ABB RAPID module: 0026CD4A

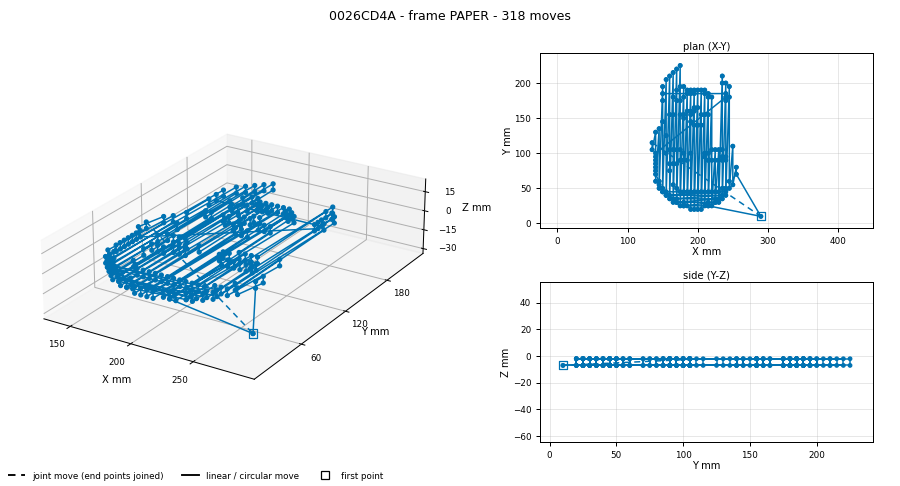
[picture p0: tool path of 0026CD4A in frame PAPER, 318 of 318 moves have a stored position in this frame; points joined in program order, loops and branches not executed]
MODULE Module1
    CONST robtarget Target_drawing_origin:=[[290,10,-2],[1,0,0,0],[0,0,0,0],[9E+09,9E+09,9E+09,9E+09,9E+09,9E+09]];


! Main procedure
PROC main()


! Clean
SetDO Do_Clean, 1;
SetDO Do_Clean, 0;
SetDO Do_Kreslit_OFF, 1;
SetDO Do_Kreslit_ON, 0;
! Draw grey
MoveJ Offs(Target_drawing_origin,0,0,-5),v100,fine,PencilHolder\WObj:=PAPER;
MoveL Offs(Target_drawing_origin,-35,60,-5),v100,fine,PencilHolder\WObj:=PAPER;
WaitRob \InPos;
MoveL Offs(Target_drawing_origin,-35,60,0),v100,fine,PencilHolder\WObj:=PAPER;
WaitRob \InPos;
SetDO Do_Kreslit_ON, 1;
SetDO Do_Kreslit_OFF, 0;
MoveL Offs(Target_drawing_origin,-35,70,0),v100,fine,PencilHolder\WObj:=PAPER;
WaitRob \InPos;
SetDO Do_Kreslit_ON, 0;
SetDO Do_Kreslit_OFF, 1;
MoveL Offs(Target_drawing_origin,-35,70,-5),v100,fine,PencilHolder\WObj:=PAPER;
WaitRob \InPos;
MoveL Offs(Target_drawing_origin,-40,45,-5),v100,fine,PencilHolder\WObj:=PAPER;
WaitRob \InPos;
MoveL Offs(Target_drawing_origin,-40,45,0),v100,fine,PencilHolder\WObj:=PAPER;
WaitRob \InPos;
SetDO Do_Kreslit_ON, 1;
SetDO Do_Kreslit_OFF, 0;
MoveL Offs(Target_drawing_origin,-40,100,0),v100,fine,PencilHolder\WObj:=PAPER;
WaitRob \InPos;
SetDO Do_Kreslit_ON, 0;
SetDO Do_Kreslit_OFF, 1;
MoveL Offs(Target_drawing_origin,-40,100,-5),v100,fine,PencilHolder\WObj:=PAPER;
WaitRob \InPos;
MoveL Offs(Target_drawing_origin,-45,40,-5),v100,fine,PencilHolder\WObj:=PAPER;
WaitRob \InPos;
MoveL Offs(Target_drawing_origin,-45,40,0),v100,fine,PencilHolder\WObj:=PAPER;
WaitRob \InPos;
SetDO Do_Kreslit_ON, 1;
SetDO Do_Kreslit_OFF, 0;
MoveL Offs(Target_drawing_origin,-45,50,0),v100,fine,PencilHolder\WObj:=PAPER;
WaitRob \InPos;
SetDO Do_Kreslit_ON, 0;
SetDO Do_Kreslit_OFF, 1;
MoveL Offs(Target_drawing_origin,-45,50,-5),v100,fine,PencilHolder\WObj:=PAPER;
WaitRob \InPos;
MoveL Offs(Target_drawing_origin,-45,170,-5),v100,fine,PencilHolder\WObj:=PAPER;
WaitRob \InPos;
MoveL Offs(Target_drawing_origin,-45,170,0),v100,fine,PencilHolder\WObj:=PAPER;
WaitRob \InPos;
SetDO Do_Kreslit_ON, 1;
SetDO Do_Kreslit_OFF, 0;
MoveL Offs(Target_drawing_origin,-45,185,0),v100,fine,PencilHolder\WObj:=PAPER;
WaitRob \InPos;
SetDO Do_Kreslit_ON, 0;
SetDO Do_Kreslit_OFF, 1;
MoveL Offs(Target_drawing_origin,-45,185,-5),v100,fine,PencilHolder\WObj:=PAPER;
WaitRob \InPos;
MoveL Offs(Target_drawing_origin,-50,30,-5),v100,fine,PencilHolder\WObj:=PAPER;
WaitRob \InPos;
MoveL Offs(Target_drawing_origin,-50,30,0),v100,fine,PencilHolder\WObj:=PAPER;
WaitRob \InPos;
SetDO Do_Kreslit_ON, 1;
SetDO Do_Kreslit_OFF, 0;
MoveL Offs(Target_drawing_origin,-50,40,0),v100,fine,PencilHolder\WObj:=PAPER;
WaitRob \InPos;
SetDO Do_Kreslit_ON, 0;
SetDO Do_Kreslit_OFF, 1;
MoveL Offs(Target_drawing_origin,-50,40,-5),v100,fine,PencilHolder\WObj:=PAPER;
WaitRob \InPos;
MoveL Offs(Target_drawing_origin,-50,80,-5),v100,fine,PencilHolder\WObj:=PAPER;
WaitRob \InPos;
MoveL Offs(Target_drawing_origin,-50,80,0),v100,fine,PencilHolder\WObj:=PAPER;
WaitRob \InPos;
SetDO Do_Kreslit_ON, 1;
SetDO Do_Kreslit_OFF, 0;
MoveL Offs(Target_drawing_origin,-50,85,0),v100,fine,PencilHolder\WObj:=PAPER;
WaitRob \InPos;
SetDO Do_Kreslit_ON, 0;
SetDO Do_Kreslit_OFF, 1;
MoveL Offs(Target_drawing_origin,-50,85,-5),v100,fine,PencilHolder\WObj:=PAPER;
WaitRob \InPos;
MoveL Offs(Target_drawing_origin,-50,165,-5),v100,fine,PencilHolder\WObj:=PAPER;
WaitRob \InPos;
MoveL Offs(Target_drawing_origin,-50,165,0),v100,fine,PencilHolder\WObj:=PAPER;
WaitRob \InPos;
SetDO Do_Kreslit_ON, 1;
SetDO Do_Kreslit_OFF, 0;
MoveL Offs(Target_drawing_origin,-50,190,0),v100,fine,PencilHolder\WObj:=PAPER;
WaitRob \InPos;
SetDO Do_Kreslit_ON, 0;
SetDO Do_Kreslit_OFF, 1;
MoveL Offs(Target_drawing_origin,-50,190,-5),v100,fine,PencilHolder\WObj:=PAPER;
WaitRob \InPos;
MoveL Offs(Target_drawing_origin,-55,25,-5),v100,fine,PencilHolder\WObj:=PAPER;
WaitRob \InPos;
MoveL Offs(Target_drawing_origin,-55,25,0),v100,fine,PencilHolder\WObj:=PAPER;
WaitRob \InPos;
SetDO Do_Kreslit_ON, 1;
SetDO Do_Kreslit_OFF, 0;
MoveL Offs(Target_drawing_origin,-55,40,0),v100,fine,PencilHolder\WObj:=PAPER;
WaitRob \InPos;
SetDO Do_Kreslit_ON, 0;
SetDO Do_Kreslit_OFF, 1;
MoveL Offs(Target_drawing_origin,-55,40,-5),v100,fine,PencilHolder\WObj:=PAPER;
WaitRob \InPos;
MoveL Offs(Target_drawing_origin,-55,80,-5),v100,fine,PencilHolder\WObj:=PAPER;
WaitRob \InPos;
MoveL Offs(Target_drawing_origin,-55,80,0),v100,fine,PencilHolder\WObj:=PAPER;
WaitRob \InPos;
SetDO Do_Kreslit_ON, 1;
SetDO Do_Kreslit_OFF, 0;
MoveL Offs(Target_drawing_origin,-55,85,0),v100,fine,PencilHolder\WObj:=PAPER;
WaitRob \InPos;
SetDO Do_Kreslit_ON, 0;
SetDO Do_Kreslit_OFF, 1;
MoveL Offs(Target_drawing_origin,-55,85,-5),v100,fine,PencilHolder\WObj:=PAPER;
WaitRob \InPos;
MoveL Offs(Target_drawing_origin,-55,95,-5),v100,fine,PencilHolder\WObj:=PAPER;
WaitRob \InPos;
MoveL Offs(Target_drawing_origin,-55,95,0),v100,fine,PencilHolder\WObj:=PAPER;
WaitRob \InPos;
SetDO Do_Kreslit_ON, 1;
SetDO Do_Kreslit_OFF, 0;
MoveL Offs(Target_drawing_origin,-55,190,0),v100,fine,PencilHolder\WObj:=PAPER;
WaitRob \InPos;
SetDO Do_Kreslit_ON, 0;
SetDO Do_Kreslit_OFF, 1;
MoveL Offs(Target_drawing_origin,-55,190,-5),v100,fine,PencilHolder\WObj:=PAPER;
WaitRob \InPos;
MoveL Offs(Target_drawing_origin,-55,200,-5),v100,fine,PencilHolder\WObj:=PAPER;
WaitRob \InPos;
MoveL Offs(Target_drawing_origin,-55,200,0),v100,fine,PencilHolder\WObj:=PAPER;
WaitRob \InPos;
SetDO Do_Kreslit_ON, 1;
SetDO Do_Kreslit_OFF, 0;
MoveL Offs(Target_drawing_origin,-60,20,0),v100,fine,PencilHolder\WObj:=PAPER;
WaitRob \InPos;
SetDO Do_Kreslit_ON, 0;
SetDO Do_Kreslit_OFF, 1;
MoveL Offs(Target_drawing_origin,-60,20,-5),v100,fine,PencilHolder\WObj:=PAPER;
WaitRob \InPos;
MoveL Offs(Target_drawing_origin,-60,35,-5),v100,fine,PencilHolder\WObj:=PAPER;
WaitRob \InPos;
MoveL Offs(Target_drawing_origin,-60,35,0),v100,fine,PencilHolder\WObj:=PAPER;
WaitRob \InPos;
SetDO Do_Kreslit_ON, 1;
SetDO Do_Kreslit_OFF, 0;
MoveL Offs(Target_drawing_origin,-60,80,0),v100,fine,PencilHolder\WObj:=PAPER;
WaitRob \InPos;
SetDO Do_Kreslit_ON, 0;
SetDO Do_Kreslit_OFF, 1;
MoveL Offs(Target_drawing_origin,-60,80,-5),v100,fine,PencilHolder\WObj:=PAPER;
WaitRob \InPos;
MoveL Offs(Target_drawing_origin,-60,95,-5),v100,fine,PencilHolder\WObj:=PAPER;
WaitRob \InPos;
MoveL Offs(Target_drawing_origin,-60,95,0),v100,fine,PencilHolder\WObj:=PAPER;
WaitRob \InPos;
SetDO Do_Kreslit_ON, 1;
SetDO Do_Kreslit_OFF, 0;
MoveL Offs(Target_drawing_origin,-65,20,0),v100,fine,PencilHolder\WObj:=PAPER;
WaitRob \InPos;
SetDO Do_Kreslit_ON, 0;
SetDO Do_Kreslit_OFF, 1;
MoveL Offs(Target_drawing_origin,-65,20,-5),v100,fine,PencilHolder\WObj:=PAPER;
WaitRob \InPos;
MoveL Offs(Target_drawing_origin,-65,35,-5),v100,fine,PencilHolder\WObj:=PAPER;
WaitRob \InPos;
MoveL Offs(Target_drawing_origin,-65,35,0),v100,fine,PencilHolder\WObj:=PAPER;
WaitRob \InPos;
SetDO Do_Kreslit_ON, 1;
SetDO Do_Kreslit_OFF, 0;
MoveL Offs(Target_drawing_origin,-65,80,0),v100,fine,PencilHolder\WObj:=PAPER;
WaitRob \InPos;
SetDO Do_Kreslit_ON, 0;
SetDO Do_Kreslit_OFF, 1;
MoveL Offs(Target_drawing_origin,-65,80,-5),v100,fine,PencilHolder\WObj:=PAPER;
WaitRob \InPos;
MoveL Offs(Target_drawing_origin,-65,95,-5),v100,fine,PencilHolder\WObj:=PAPER;
WaitRob \InPos;
MoveL Offs(Target_drawing_origin,-65,95,0),v100,fine,PencilHolder\WObj:=PAPER;
WaitRob \InPos;
SetDO Do_Kreslit_ON, 1;
SetDO Do_Kreslit_OFF, 0;
MoveL Offs(Target_drawing_origin,-70,15,0),v100,fine,PencilHolder\WObj:=PAPER;
WaitRob \InPos;
SetDO Do_Kreslit_ON, 0;
SetDO Do_Kreslit_OFF, 1;
MoveL Offs(Target_drawing_origin,-70,15,-5),v100,fine,PencilHolder\WObj:=PAPER;
WaitRob \InPos;
MoveL Offs(Target_drawing_origin,-70,35,-5),v100,fine,PencilHolder\WObj:=PAPER;
WaitRob \InPos;
MoveL Offs(Target_drawing_origin,-70,35,0),v100,fine,PencilHolder\WObj:=PAPER;
WaitRob \InPos;
SetDO Do_Kreslit_ON, 1;
SetDO Do_Kreslit_OFF, 0;
MoveL Offs(Target_drawing_origin,-70,80,0),v100,fine,PencilHolder\WObj:=PAPER;
WaitRob \InPos;
SetDO Do_Kreslit_ON, 0;
SetDO Do_Kreslit_OFF, 1;
MoveL Offs(Target_drawing_origin,-70,80,-5),v100,fine,PencilHolder\WObj:=PAPER;
WaitRob \InPos;
MoveL Offs(Target_drawing_origin,-70,95,-5),v100,fine,PencilHolder\WObj:=PAPER;
WaitRob \InPos;
MoveL Offs(Target_drawing_origin,-70,95,0),v100,fine,PencilHolder\WObj:=PAPER;
WaitRob \InPos;
SetDO Do_Kreslit_ON, 1;
SetDO Do_Kreslit_OFF, 0;
MoveL Offs(Target_drawing_origin,-70,170,0),v100,fine,PencilHolder\WObj:=PAPER;
WaitRob \InPos;
SetDO Do_Kreslit_ON, 0;
SetDO Do_Kreslit_OFF, 1;
MoveL Offs(Target_drawing_origin,-70,170,-5),v100,fine,PencilHolder\WObj:=PAPER;
WaitRob \InPos;
MoveL Offs(Target_drawing_origin,-75,15,-5),v100,fine,PencilHolder\WObj:=PAPER;
WaitRob \InPos;
MoveL Offs(Target_drawing_origin,-75,15,0),v100,fine,PencilHolder\WObj:=PAPER;
WaitRob \InPos;
SetDO Do_Kreslit_ON, 1;
SetDO Do_Kreslit_OFF, 0;
MoveL Offs(Target_drawing_origin,-75,35,0),v100,fine,PencilHolder\WObj:=PAPER;
WaitRob \InPos;
SetDO Do_Kreslit_ON, 0;
SetDO Do_Kreslit_OFF, 1;
MoveL Offs(Target_drawing_origin,-75,35,-5),v100,fine,PencilHolder\WObj:=PAPER;
WaitRob \InPos;
MoveL Offs(Target_drawing_origin,-75,80,-5),v100,fine,PencilHolder\WObj:=PAPER;
WaitRob \InPos;
MoveL Offs(Target_drawing_origin,-75,80,0),v100,fine,PencilHolder\WObj:=PAPER;
WaitRob \InPos;
SetDO Do_Kreslit_ON, 1;
SetDO Do_Kreslit_OFF, 0;
MoveL Offs(Target_drawing_origin,-75,90,0),v100,fine,PencilHolder\WObj:=PAPER;
WaitRob \InPos;
SetDO Do_Kreslit_ON, 0;
SetDO Do_Kreslit_OFF, 1;
MoveL Offs(Target_drawing_origin,-75,90,-5),v100,fine,PencilHolder\WObj:=PAPER;
WaitRob \InPos;
MoveL Offs(Target_drawing_origin,-75,145,-5),v100,fine,PencilHolder\WObj:=PAPER;
WaitRob \InPos;
MoveL Offs(Target_drawing_origin,-75,145,0),v100,fine,PencilHolder\WObj:=PAPER;
WaitRob \InPos;
SetDO Do_Kreslit_ON, 1;
SetDO Do_Kreslit_OFF, 0;
MoveL Offs(Target_drawing_origin,-75,170,0),v100,fine,PencilHolder\WObj:=PAPER;
WaitRob \InPos;
SetDO Do_Kreslit_ON, 0;
SetDO Do_Kreslit_OFF, 1;
MoveL Offs(Target_drawing_origin,-75,170,-5),v100,fine,PencilHolder\WObj:=PAPER;
WaitRob \InPos;
MoveL Offs(Target_drawing_origin,-75,175,-5),v100,fine,PencilHolder\WObj:=PAPER;
WaitRob \InPos;
MoveL Offs(Target_drawing_origin,-75,175,0),v100,fine,PencilHolder\WObj:=PAPER;
WaitRob \InPos;
SetDO Do_Kreslit_ON, 1;
SetDO Do_Kreslit_OFF, 0;
MoveL Offs(Target_drawing_origin,-80,15,0),v100,fine,PencilHolder\WObj:=PAPER;
WaitRob \InPos;
SetDO Do_Kreslit_ON, 0;
SetDO Do_Kreslit_OFF, 1;
MoveL Offs(Target_drawing_origin,-80,15,-5),v100,fine,PencilHolder\WObj:=PAPER;
WaitRob \InPos;
MoveL Offs(Target_drawing_origin,-80,35,-5),v100,fine,PencilHolder\WObj:=PAPER;
WaitRob \InPos;
MoveL Offs(Target_drawing_origin,-80,35,0),v100,fine,PencilHolder\WObj:=PAPER;
WaitRob \InPos;
SetDO Do_Kreslit_ON, 1;
SetDO Do_Kreslit_OFF, 0;
MoveL Offs(Target_drawing_origin,-80,85,0),v100,fine,PencilHolder\WObj:=PAPER;
WaitRob \InPos;
SetDO Do_Kreslit_ON, 0;
SetDO Do_Kreslit_OFF, 1;
MoveL Offs(Target_drawing_origin,-80,85,-5),v100,fine,PencilHolder\WObj:=PAPER;
WaitRob \InPos;
MoveL Offs(Target_drawing_origin,-80,90,-5),v100,fine,PencilHolder\WObj:=PAPER;
WaitRob \InPos;
MoveL Offs(Target_drawing_origin,-80,90,0),v100,fine,PencilHolder\WObj:=PAPER;
WaitRob \InPos;
SetDO Do_Kreslit_ON, 1;
SetDO Do_Kreslit_OFF, 0;
MoveL Offs(Target_drawing_origin,-80,145,0),v100,fine,PencilHolder\WObj:=PAPER;
WaitRob \InPos;
SetDO Do_Kreslit_ON, 0;
SetDO Do_Kreslit_OFF, 1;
MoveL Offs(Target_drawing_origin,-80,145,-5),v100,fine,PencilHolder\WObj:=PAPER;
WaitRob \InPos;
MoveL Offs(Target_drawing_origin,-80,175,-5),v100,fine,PencilHolder\WObj:=PAPER;
WaitRob \InPos;
MoveL Offs(Target_drawing_origin,-80,175,0),v100,fine,PencilHolder\WObj:=PAPER;
WaitRob \InPos;
SetDO Do_Kreslit_ON, 1;
SetDO Do_Kreslit_OFF, 0;
MoveL Offs(Target_drawing_origin,-80,180,0),v100,fine,PencilHolder\WObj:=PAPER;
WaitRob \InPos;
SetDO Do_Kreslit_ON, 0;
SetDO Do_Kreslit_OFF, 1;
MoveL Offs(Target_drawing_origin,-80,180,-5),v100,fine,PencilHolder\WObj:=PAPER;
WaitRob \InPos;
MoveL Offs(Target_drawing_origin,-85,10,-5),v100,fine,PencilHolder\WObj:=PAPER;
WaitRob \InPos;
MoveL Offs(Target_drawing_origin,-85,10,0),v100,fine,PencilHolder\WObj:=PAPER;
WaitRob \InPos;
SetDO Do_Kreslit_ON, 1;
SetDO Do_Kreslit_OFF, 0;
MoveL Offs(Target_drawing_origin,-85,35,0),v100,fine,PencilHolder\WObj:=PAPER;
WaitRob \InPos;
SetDO Do_Kreslit_ON, 0;
SetDO Do_Kreslit_OFF, 1;
MoveL Offs(Target_drawing_origin,-85,35,-5),v100,fine,PencilHolder\WObj:=PAPER;
WaitRob \InPos;
MoveL Offs(Target_drawing_origin,-85,130,-5),v100,fine,PencilHolder\WObj:=PAPER;
WaitRob \InPos;
MoveL Offs(Target_drawing_origin,-85,130,0),v100,fine,PencilHolder\WObj:=PAPER;
WaitRob \InPos;
SetDO Do_Kreslit_ON, 1;
SetDO Do_Kreslit_OFF, 0;
MoveL Offs(Target_drawing_origin,-85,145,0),v100,fine,PencilHolder\WObj:=PAPER;
WaitRob \InPos;
SetDO Do_Kreslit_ON, 0;
SetDO Do_Kreslit_OFF, 1;
MoveL Offs(Target_drawing_origin,-85,145,-5),v100,fine,PencilHolder\WObj:=PAPER;
WaitRob \InPos;
MoveL Offs(Target_drawing_origin,-85,180,-5),v100,fine,PencilHolder\WObj:=PAPER;
WaitRob \InPos;
MoveL Offs(Target_drawing_origin,-85,180,0),v100,fine,PencilHolder\WObj:=PAPER;
WaitRob \InPos;
SetDO Do_Kreslit_ON, 1;
SetDO Do_Kreslit_OFF, 0;
MoveL Offs(Target_drawing_origin,-90,10,0),v100,fine,PencilHolder\WObj:=PAPER;
WaitRob \InPos;
SetDO Do_Kreslit_ON, 0;
SetDO Do_Kreslit_OFF, 1;
MoveL Offs(Target_drawing_origin,-90,10,-5),v100,fine,PencilHolder\WObj:=PAPER;
WaitRob \InPos;
MoveL Offs(Target_drawing_origin,-90,35,-5),v100,fine,PencilHolder\WObj:=PAPER;
WaitRob \InPos;
MoveL Offs(Target_drawing_origin,-90,35,0),v100,fine,PencilHolder\WObj:=PAPER;
WaitRob \InPos;
SetDO Do_Kreslit_ON, 1;
SetDO Do_Kreslit_OFF, 0;
MoveL Offs(Target_drawing_origin,-90,130,0),v100,fine,PencilHolder\WObj:=PAPER;
WaitRob \InPos;
SetDO Do_Kreslit_ON, 0;
SetDO Do_Kreslit_OFF, 1;
MoveL Offs(Target_drawing_origin,-90,130,-5),v100,fine,PencilHolder\WObj:=PAPER;
WaitRob \InPos;
MoveL Offs(Target_drawing_origin,-90,155,-5),v100,fine,PencilHolder\WObj:=PAPER;
WaitRob \InPos;
MoveL Offs(Target_drawing_origin,-90,155,0),v100,fine,PencilHolder\WObj:=PAPER;
WaitRob \InPos;
SetDO Do_Kreslit_ON, 1;
SetDO Do_Kreslit_OFF, 0;
MoveL Offs(Target_drawing_origin,-90,180,0),v100,fine,PencilHolder\WObj:=PAPER;
WaitRob \InPos;
SetDO Do_Kreslit_ON, 0;
SetDO Do_Kreslit_OFF, 1;
MoveL Offs(Target_drawing_origin,-90,180,-5),v100,fine,PencilHolder\WObj:=PAPER;
WaitRob \InPos;
MoveL Offs(Target_drawing_origin,-95,10,-5),v100,fine,PencilHolder\WObj:=PAPER;
WaitRob \InPos;
MoveL Offs(Target_drawing_origin,-95,10,0),v100,fine,PencilHolder\WObj:=PAPER;
WaitRob \InPos;
SetDO Do_Kreslit_ON, 1;
SetDO Do_Kreslit_OFF, 0;
MoveL Offs(Target_drawing_origin,-95,35,0),v100,fine,PencilHolder\WObj:=PAPER;
WaitRob \InPos;
SetDO Do_Kreslit_ON, 0;
SetDO Do_Kreslit_OFF, 1;
MoveL Offs(Target_drawing_origin,-95,35,-5),v100,fine,PencilHolder\WObj:=PAPER;
WaitRob \InPos;
MoveL Offs(Target_drawing_origin,-95,130,-5),v100,fine,PencilHolder\WObj:=PAPER;
WaitRob \InPos;
MoveL Offs(Target_drawing_origin,-95,130,0),v100,fine,PencilHolder\WObj:=PAPER;
WaitRob \InPos;
SetDO Do_Kreslit_ON, 1;
SetDO Do_Kreslit_OFF, 0;
MoveL Offs(Target_drawing_origin,-95,150,0),v100,fine,PencilHolder\WObj:=PAPER;
WaitRob \InPos;
SetDO Do_Kreslit_ON, 0;
SetDO Do_Kreslit_OFF, 1;
MoveL Offs(Target_drawing_origin,-95,150,-5),v100,fine,PencilHolder\WObj:=PAPER;
WaitRob \InPos;
MoveL Offs(Target_drawing_origin,-95,155,-5),v100,fine,PencilHolder\WObj:=PAPER;
WaitRob \InPos;
MoveL Offs(Target_drawing_origin,-95,155,0),v100,fine,PencilHolder\WObj:=PAPER;
WaitRob \InPos;
SetDO Do_Kreslit_ON, 1;
SetDO Do_Kreslit_OFF, 0;
MoveL Offs(Target_drawing_origin,-95,175,0),v100,fine,PencilHolder\WObj:=PAPER;
WaitRob \InPos;
SetDO Do_Kreslit_ON, 0;
SetDO Do_Kreslit_OFF, 1;
MoveL Offs(Target_drawing_origin,-95,175,-5),v100,fine,PencilHolder\WObj:=PAPER;
WaitRob \InPos;
MoveL Offs(Target_drawing_origin,-95,180,-5),v100,fine,PencilHolder\WObj:=PAPER;
WaitRob \InPos;
MoveL Offs(Target_drawing_origin,-95,180,0),v100,fine,PencilHolder\WObj:=PAPER;
WaitRob \InPos;
SetDO Do_Kreslit_ON, 1;
SetDO Do_Kreslit_OFF, 0;
MoveL Offs(Target_drawing_origin,-100,10,0),v100,fine,PencilHolder\WObj:=PAPER;
WaitRob \InPos;
SetDO Do_Kreslit_ON, 0;
SetDO Do_Kreslit_OFF, 1;
MoveL Offs(Target_drawing_origin,-100,10,-5),v100,fine,PencilHolder\WObj:=PAPER;
WaitRob \InPos;
MoveL Offs(Target_drawing_origin,-100,35,-5),v100,fine,PencilHolder\WObj:=PAPER;
WaitRob \InPos;
MoveL Offs(Target_drawing_origin,-100,35,0),v100,fine,PencilHolder\WObj:=PAPER;
WaitRob \InPos;
SetDO Do_Kreslit_ON, 1;
SetDO Do_Kreslit_OFF, 0;
MoveL Offs(Target_drawing_origin,-100,90,0),v100,fine,PencilHolder\WObj:=PAPER;
WaitRob \InPos;
SetDO Do_Kreslit_ON, 0;
SetDO Do_Kreslit_OFF, 1;
MoveL Offs(Target_drawing_origin,-100,90,-5),v100,fine,PencilHolder\WObj:=PAPER;
WaitRob \InPos;
MoveL Offs(Target_drawing_origin,-100,135,-5),v100,fine,PencilHolder\WObj:=PAPER;
WaitRob \InPos;
MoveL Offs(Target_drawing_origin,-100,135,0),v100,fine,PencilHolder\WObj:=PAPER;
WaitRob \InPos;
SetDO Do_Kreslit_ON, 1;
SetDO Do_Kreslit_OFF, 0;
MoveL Offs(Target_drawing_origin,-100,145,0),v100,fine,PencilHolder\WObj:=PAPER;
WaitRob \InPos;
SetDO Do_Kreslit_ON, 0;
SetDO Do_Kreslit_OFF, 1;
MoveL Offs(Target_drawing_origin,-100,145,-5),v100,fine,PencilHolder\WObj:=PAPER;
WaitRob \InPos;
MoveL Offs(Target_drawing_origin,-100,150,-5),v100,fine,PencilHolder\WObj:=PAPER;
WaitRob \InPos;
MoveL Offs(Target_drawing_origin,-100,150,0),v100,fine,PencilHolder\WObj:=PAPER;
WaitRob \InPos;
SetDO Do_Kreslit_ON, 1;
SetDO Do_Kreslit_OFF, 0;
MoveL Offs(Target_drawing_origin,-100,175,0),v100,fine,PencilHolder\WObj:=PAPER;
WaitRob \InPos;
SetDO Do_Kreslit_ON, 0;
SetDO Do_Kreslit_OFF, 1;
MoveL Offs(Target_drawing_origin,-100,175,-5),v100,fine,PencilHolder\WObj:=PAPER;
WaitRob \InPos;
MoveL Offs(Target_drawing_origin,-100,180,-5),v100,fine,PencilHolder\WObj:=PAPER;
WaitRob \InPos;
MoveL Offs(Target_drawing_origin,-100,180,0),v100,fine,PencilHolder\WObj:=PAPER;
WaitRob \InPos;
SetDO Do_Kreslit_ON, 1;
SetDO Do_Kreslit_OFF, 0;
MoveL Offs(Target_drawing_origin,-105,15,0),v100,fine,PencilHolder\WObj:=PAPER;
WaitRob \InPos;
SetDO Do_Kreslit_ON, 0;
SetDO Do_Kreslit_OFF, 1;
MoveL Offs(Target_drawing_origin,-105,15,-5),v100,fine,PencilHolder\WObj:=PAPER;
WaitRob \InPos;
MoveL Offs(Target_drawing_origin,-105,35,-5),v100,fine,PencilHolder\WObj:=PAPER;
WaitRob \InPos;
MoveL Offs(Target_drawing_origin,-105,35,0),v100,fine,PencilHolder\WObj:=PAPER;
WaitRob \InPos;
SetDO Do_Kreslit_ON, 1;
SetDO Do_Kreslit_OFF, 0;
MoveL Offs(Target_drawing_origin,-105,80,0),v100,fine,PencilHolder\WObj:=PAPER;
WaitRob \InPos;
SetDO Do_Kreslit_ON, 0;
SetDO Do_Kreslit_OFF, 1;
MoveL Offs(Target_drawing_origin,-105,80,-5),v100,fine,PencilHolder\WObj:=PAPER;
WaitRob \InPos;
MoveL Offs(Target_drawing_origin,-105,150,-5),v100,fine,PencilHolder\WObj:=PAPER;
WaitRob \InPos;
MoveL Offs(Target_drawing_origin,-105,150,0),v100,fine,PencilHolder\WObj:=PAPER;
WaitRob \InPos;
SetDO Do_Kreslit_ON, 1;
SetDO Do_Kreslit_OFF, 0;
MoveL Offs(Target_drawing_origin,-105,175,0),v100,fine,PencilHolder\WObj:=PAPER;
WaitRob \InPos;
SetDO Do_Kreslit_ON, 0;
SetDO Do_Kreslit_OFF, 1;
MoveL Offs(Target_drawing_origin,-105,175,-5),v100,fine,PencilHolder\WObj:=PAPER;
WaitRob \InPos;
MoveL Offs(Target_drawing_origin,-105,180,-5),v100,fine,PencilHolder\WObj:=PAPER;
WaitRob \InPos;
MoveL Offs(Target_drawing_origin,-105,180,0),v100,fine,PencilHolder\WObj:=PAPER;
WaitRob \InPos;
SetDO Do_Kreslit_ON, 1;
SetDO Do_Kreslit_OFF, 0;
MoveL Offs(Target_drawing_origin,-110,15,0),v100,fine,PencilHolder\WObj:=PAPER;
WaitRob \InPos;
SetDO Do_Kreslit_ON, 0;
SetDO Do_Kreslit_OFF, 1;
MoveL Offs(Target_drawing_origin,-110,15,-5),v100,fine,PencilHolder\WObj:=PAPER;
WaitRob \InPos;
MoveL Offs(Target_drawing_origin,-110,35,-5),v100,fine,PencilHolder\WObj:=PAPER;
WaitRob \InPos;
MoveL Offs(Target_drawing_origin,-110,35,0),v100,fine,PencilHolder\WObj:=PAPER;
WaitRob \InPos;
SetDO Do_Kreslit_ON, 1;
SetDO Do_Kreslit_OFF, 0;
MoveL Offs(Target_drawing_origin,-110,80,0),v100,fine,PencilHolder\WObj:=PAPER;
WaitRob \InPos;
SetDO Do_Kreslit_ON, 0;
SetDO Do_Kreslit_OFF, 1;
MoveL Offs(Target_drawing_origin,-110,80,-5),v100,fine,PencilHolder\WObj:=PAPER;
WaitRob \InPos;
MoveL Offs(Target_drawing_origin,-110,90,-5),v100,fine,PencilHolder\WObj:=PAPER;
WaitRob \InPos;
MoveL Offs(Target_drawing_origin,-110,90,0),v100,fine,PencilHolder\WObj:=PAPER;
WaitRob \InPos;
SetDO Do_Kreslit_ON, 1;
SetDO Do_Kreslit_OFF, 0;
MoveL Offs(Target_drawing_origin,-110,140,0),v100,fine,PencilHolder\WObj:=PAPER;
WaitRob \InPos;
SetDO Do_Kreslit_ON, 0;
SetDO Do_Kreslit_OFF, 1;
MoveL Offs(Target_drawing_origin,-110,140,-5),v100,fine,PencilHolder\WObj:=PAPER;
WaitRob \InPos;
MoveL Offs(Target_drawing_origin,-110,145,-5),v100,fine,PencilHolder\WObj:=PAPER;
WaitRob \InPos;
MoveL Offs(Target_drawing_origin,-110,145,0),v100,fine,PencilHolder\WObj:=PAPER;
WaitRob \InPos;
SetDO Do_Kreslit_ON, 1;
SetDO Do_Kreslit_OFF, 0;
MoveL Offs(Target_drawing_origin,-110,170,0),v100,fine,PencilHolder\WObj:=PAPER;
WaitRob \InPos;
SetDO Do_Kreslit_ON, 0;
SetDO Do_Kreslit_OFF, 1;
MoveL Offs(Target_drawing_origin,-110,170,-5),v100,fine,PencilHolder\WObj:=PAPER;
WaitRob \InPos;
MoveL Offs(Target_drawing_origin,-110,185,-5),v100,fine,PencilHolder\WObj:=PAPER;
WaitRob \InPos;
MoveL Offs(Target_drawing_origin,-110,185,0),v100,fine,PencilHolder\WObj:=PAPER;
WaitRob \InPos;
SetDO Do_Kreslit_ON, 1;
SetDO Do_Kreslit_OFF, 0;
MoveL Offs(Target_drawing_origin,-115,15,0),v100,fine,PencilHolder\WObj:=PAPER;
WaitRob \InPos;
SetDO Do_Kreslit_ON, 0;
SetDO Do_Kreslit_OFF, 1;
MoveL Offs(Target_drawing_origin,-115,15,-5),v100,fine,PencilHolder\WObj:=PAPER;
WaitRob \InPos;
MoveL Offs(Target_drawing_origin,-115,35,-5),v100,fine,PencilHolder\WObj:=PAPER;
WaitRob \InPos;
MoveL Offs(Target_drawing_origin,-115,35,0),v100,fine,PencilHolder\WObj:=PAPER;
WaitRob \InPos;
SetDO Do_Kreslit_ON, 1;
SetDO Do_Kreslit_OFF, 0;
MoveL Offs(Target_drawing_origin,-115,80,0),v100,fine,PencilHolder\WObj:=PAPER;
WaitRob \InPos;
SetDO Do_Kreslit_ON, 0;
SetDO Do_Kreslit_OFF, 1;
MoveL Offs(Target_drawing_origin,-115,80,-5),v100,fine,PencilHolder\WObj:=PAPER;
WaitRob \InPos;
MoveL Offs(Target_drawing_origin,-115,95,-5),v100,fine,PencilHolder\WObj:=PAPER;
WaitRob \InPos;
MoveL Offs(Target_drawing_origin,-115,95,0),v100,fine,PencilHolder\WObj:=PAPER;
WaitRob \InPos;
SetDO Do_Kreslit_ON, 1;
SetDO Do_Kreslit_OFF, 0;
MoveL Offs(Target_drawing_origin,-115,145,0),v100,fine,PencilHolder\WObj:=PAPER;
WaitRob \InPos;
SetDO Do_Kreslit_ON, 0;
SetDO Do_Kreslit_OFF, 1;
MoveL Offs(Target_drawing_origin,-115,145,-5),v100,fine,PencilHolder\WObj:=PAPER;
WaitRob \InPos;
MoveL Offs(Target_drawing_origin,-115,165,-5),v100,fine,PencilHolder\WObj:=PAPER;
WaitRob \InPos;
MoveL Offs(Target_drawing_origin,-115,165,0),v100,fine,PencilHolder\WObj:=PAPER;
WaitRob \InPos;
SetDO Do_Kreslit_ON, 1;
SetDO Do_Kreslit_OFF, 0;
MoveL Offs(Target_drawing_origin,-115,185,0),v100,fine,PencilHolder\WObj:=PAPER;
WaitRob \InPos;
SetDO Do_Kreslit_ON, 0;
SetDO Do_Kreslit_OFF, 1;
MoveL Offs(Target_drawing_origin,-115,185,-5),v100,fine,PencilHolder\WObj:=PAPER;
WaitRob \InPos;
MoveL Offs(Target_drawing_origin,-115,215,-5),v100,fine,PencilHolder\WObj:=PAPER;
WaitRob \InPos;
MoveL Offs(Target_drawing_origin,-115,215,0),v100,fine,PencilHolder\WObj:=PAPER;
WaitRob \InPos;
SetDO Do_Kreslit_ON, 1;
SetDO Do_Kreslit_OFF, 0;
MoveL Offs(Target_drawing_origin,-120,20,0),v100,fine,PencilHolder\WObj:=PAPER;
WaitRob \InPos;
SetDO Do_Kreslit_ON, 0;
SetDO Do_Kreslit_OFF, 1;
MoveL Offs(Target_drawing_origin,-120,20,-5),v100,fine,PencilHolder\WObj:=PAPER;
WaitRob \InPos;
MoveL Offs(Target_drawing_origin,-120,40,-5),v100,fine,PencilHolder\WObj:=PAPER;
WaitRob \InPos;
MoveL Offs(Target_drawing_origin,-120,40,0),v100,fine,PencilHolder\WObj:=PAPER;
WaitRob \InPos;
SetDO Do_Kreslit_ON, 1;
SetDO Do_Kreslit_OFF, 0;
MoveL Offs(Target_drawing_origin,-120,75,0),v100,fine,PencilHolder\WObj:=PAPER;
WaitRob \InPos;
SetDO Do_Kreslit_ON, 0;
SetDO Do_Kreslit_OFF, 1;
MoveL Offs(Target_drawing_origin,-120,75,-5),v100,fine,PencilHolder\WObj:=PAPER;
WaitRob \InPos;
MoveL Offs(Target_drawing_origin,-120,95,-5),v100,fine,PencilHolder\WObj:=PAPER;
WaitRob \InPos;
MoveL Offs(Target_drawing_origin,-120,95,0),v100,fine,PencilHolder\WObj:=PAPER;
WaitRob \InPos;
SetDO Do_Kreslit_ON, 1;
SetDO Do_Kreslit_OFF, 0;
MoveL Offs(Target_drawing_origin,-120,165,0),v100,fine,PencilHolder\WObj:=PAPER;
WaitRob \InPos;
SetDO Do_Kreslit_ON, 0;
SetDO Do_Kreslit_OFF, 1;
MoveL Offs(Target_drawing_origin,-120,165,-5),v100,fine,PencilHolder\WObj:=PAPER;
WaitRob \InPos;
MoveL Offs(Target_drawing_origin,-120,180,-5),v100,fine,PencilHolder\WObj:=PAPER;
WaitRob \InPos;
MoveL Offs(Target_drawing_origin,-120,180,0),v100,fine,PencilHolder\WObj:=PAPER;
WaitRob \InPos;
SetDO Do_Kreslit_ON, 1;
SetDO Do_Kreslit_OFF, 0;
MoveL Offs(Target_drawing_origin,-120,210,0),v100,fine,PencilHolder\WObj:=PAPER;
WaitRob \InPos;
SetDO Do_Kreslit_ON, 0;
SetDO Do_Kreslit_OFF, 1;
MoveL Offs(Target_drawing_origin,-120,210,-5),v100,fine,PencilHolder\WObj:=PAPER;
WaitRob \InPos;
MoveL Offs(Target_drawing_origin,-125,20,-5),v100,fine,PencilHolder\WObj:=PAPER;
WaitRob \InPos;
MoveL Offs(Target_drawing_origin,-125,20,0),v100,fine,PencilHolder\WObj:=PAPER;
WaitRob \InPos;
SetDO Do_Kreslit_ON, 1;
SetDO Do_Kreslit_OFF, 0;
MoveL Offs(Target_drawing_origin,-125,45,0),v100,fine,PencilHolder\WObj:=PAPER;
WaitRob \InPos;
SetDO Do_Kreslit_ON, 0;
SetDO Do_Kreslit_OFF, 1;
MoveL Offs(Target_drawing_origin,-125,45,-5),v100,fine,PencilHolder\WObj:=PAPER;
WaitRob \InPos;
MoveL Offs(Target_drawing_origin,-125,75,-5),v100,fine,PencilHolder\WObj:=PAPER;
WaitRob \InPos;
MoveL Offs(Target_drawing_origin,-125,75,0),v100,fine,PencilHolder\WObj:=PAPER;
WaitRob \InPos;
SetDO Do_Kreslit_ON, 1;
SetDO Do_Kreslit_OFF, 0;
MoveL Offs(Target_drawing_origin,-125,95,0),v100,fine,PencilHolder\WObj:=PAPER;
WaitRob \InPos;
SetDO Do_Kreslit_ON, 0;
SetDO Do_Kreslit_OFF, 1;
MoveL Offs(Target_drawing_origin,-125,95,-5),v100,fine,PencilHolder\WObj:=PAPER;
WaitRob \InPos;
MoveL Offs(Target_drawing_origin,-125,145,-5),v100,fine,PencilHolder\WObj:=PAPER;
WaitRob \InPos;
MoveL Offs(Target_drawing_origin,-125,145,0),v100,fine,PencilHolder\WObj:=PAPER;
WaitRob \InPos;
SetDO Do_Kreslit_ON, 1;
SetDO Do_Kreslit_OFF, 0;
MoveL Offs(Target_drawing_origin,-125,170,0),v100,fine,PencilHolder\WObj:=PAPER;
WaitRob \InPos;
SetDO Do_Kreslit_ON, 0;
SetDO Do_Kreslit_OFF, 1;
MoveL Offs(Target_drawing_origin,-125,170,-5),v100,fine,PencilHolder\WObj:=PAPER;
WaitRob \InPos;
MoveL Offs(Target_drawing_origin,-125,205,-5),v100,fine,PencilHolder\WObj:=PAPER;
WaitRob \InPos;
MoveL Offs(Target_drawing_origin,-125,205,0),v100,fine,PencilHolder\WObj:=PAPER;
WaitRob \InPos;
SetDO Do_Kreslit_ON, 1;
SetDO Do_Kreslit_OFF, 0;
MoveL Offs(Target_drawing_origin,-130,25,0),v100,fine,PencilHolder\WObj:=PAPER;
WaitRob \InPos;
SetDO Do_Kreslit_ON, 0;
SetDO Do_Kreslit_OFF, 1;
MoveL Offs(Target_drawing_origin,-130,25,-5),v100,fine,PencilHolder\WObj:=PAPER;
WaitRob \InPos;
MoveL Offs(Target_drawing_origin,-130,65,-5),v100,fine,PencilHolder\WObj:=PAPER;
WaitRob \InPos;
MoveL Offs(Target_drawing_origin,-130,65,0),v100,fine,PencilHolder\WObj:=PAPER;
WaitRob \InPos;
SetDO Do_Kreslit_ON, 1;
SetDO Do_Kreslit_OFF, 0;
MoveL Offs(Target_drawing_origin,-130,75,0),v100,fine,PencilHolder\WObj:=PAPER;
WaitRob \InPos;
SetDO Do_Kreslit_ON, 0;
SetDO Do_Kreslit_OFF, 1;
MoveL Offs(Target_drawing_origin,-130,75,-5),v100,fine,PencilHolder\WObj:=PAPER;
WaitRob \InPos;
MoveL Offs(Target_drawing_origin,-130,95,-5),v100,fine,PencilHolder\WObj:=PAPER;
WaitRob \InPos;
MoveL Offs(Target_drawing_origin,-130,95,0),v100,fine,PencilHolder\WObj:=PAPER;
WaitRob \InPos;
SetDO Do_Kreslit_ON, 1;
SetDO Do_Kreslit_OFF, 0;
MoveL Offs(Target_drawing_origin,-130,145,0),v100,fine,PencilHolder\WObj:=PAPER;
WaitRob \InPos;
SetDO Do_Kreslit_ON, 0;
SetDO Do_Kreslit_OFF, 1;
MoveL Offs(Target_drawing_origin,-130,145,-5),v100,fine,PencilHolder\WObj:=PAPER;
WaitRob \InPos;
MoveL Offs(Target_drawing_origin,-130,200,-5),v100,fine,PencilHolder\WObj:=PAPER;
WaitRob \InPos;
MoveL Offs(Target_drawing_origin,-130,200,0),v100,fine,PencilHolder\WObj:=PAPER;
WaitRob \InPos;
SetDO Do_Kreslit_ON, 1;
SetDO Do_Kreslit_OFF, 0;
MoveL Offs(Target_drawing_origin,-135,30,0),v100,fine,PencilHolder\WObj:=PAPER;
WaitRob \InPos;
SetDO Do_Kreslit_ON, 0;
SetDO Do_Kreslit_OFF, 1;
MoveL Offs(Target_drawing_origin,-135,30,-5),v100,fine,PencilHolder\WObj:=PAPER;
WaitRob \InPos;
MoveL Offs(Target_drawing_origin,-135,90,-5),v100,fine,PencilHolder\WObj:=PAPER;
WaitRob \InPos;
MoveL Offs(Target_drawing_origin,-135,90,0),v100,fine,PencilHolder\WObj:=PAPER;
WaitRob \InPos;
SetDO Do_Kreslit_ON, 1;
SetDO Do_Kreslit_OFF, 0;
MoveL Offs(Target_drawing_origin,-135,115,0),v100,fine,PencilHolder\WObj:=PAPER;
WaitRob \InPos;
SetDO Do_Kreslit_ON, 0;
SetDO Do_Kreslit_OFF, 1;
MoveL Offs(Target_drawing_origin,-135,115,-5),v100,fine,PencilHolder\WObj:=PAPER;
WaitRob \InPos;
MoveL Offs(Target_drawing_origin,-135,195,-5),v100,fine,PencilHolder\WObj:=PAPER;
WaitRob \InPos;
MoveL Offs(Target_drawing_origin,-135,195,0),v100,fine,PencilHolder\WObj:=PAPER;
WaitRob \InPos;
SetDO Do_Kreslit_ON, 1;
SetDO Do_Kreslit_OFF, 0;
MoveL Offs(Target_drawing_origin,-140,35,0),v100,fine,PencilHolder\WObj:=PAPER;
WaitRob \InPos;
SetDO Do_Kreslit_ON, 0;
SetDO Do_Kreslit_OFF, 1;
MoveL Offs(Target_drawing_origin,-140,35,-5),v100,fine,PencilHolder\WObj:=PAPER;
WaitRob \InPos;
MoveL Offs(Target_drawing_origin,-140,135,-5),v100,fine,PencilHolder\WObj:=PAPER;
WaitRob \InPos;
MoveL Offs(Target_drawing_origin,-140,135,0),v100,fine,PencilHolder\WObj:=PAPER;
WaitRob \InPos;
SetDO Do_Kreslit_ON, 1;
SetDO Do_Kreslit_OFF, 0;
MoveL Offs(Target_drawing_origin,-140,165,0),v100,fine,PencilHolder\WObj:=PAPER;
WaitRob \InPos;
SetDO Do_Kreslit_ON, 0;
SetDO Do_Kreslit_OFF, 1;
MoveL Offs(Target_drawing_origin,-140,165,-5),v100,fine,PencilHolder\WObj:=PAPER;
WaitRob \InPos;
MoveL Offs(Target_drawing_origin,-140,185,-5),v100,fine,PencilHolder\WObj:=PAPER;
WaitRob \InPos;
MoveL Offs(Target_drawing_origin,-140,185,0),v100,fine,PencilHolder\WObj:=PAPER;
WaitRob \InPos;
SetDO Do_Kreslit_ON, 1;
SetDO Do_Kreslit_OFF, 0;
MoveL Offs(Target_drawing_origin,-145,40,0),v100,fine,PencilHolder\WObj:=PAPER;
WaitRob \InPos;
SetDO Do_Kreslit_ON, 0;
SetDO Do_Kreslit_OFF, 1;
MoveL Offs(Target_drawing_origin,-145,40,-5),v100,fine,PencilHolder\WObj:=PAPER;
WaitRob \InPos;
MoveL Offs(Target_drawing_origin,-145,125,-5),v100,fine,PencilHolder\WObj:=PAPER;
WaitRob \InPos;
MoveL Offs(Target_drawing_origin,-145,125,0),v100,fine,PencilHolder\WObj:=PAPER;
WaitRob \InPos;
SetDO Do_Kreslit_ON, 1;
SetDO Do_Kreslit_OFF, 0;
MoveL Offs(Target_drawing_origin,-150,50,0),v100,fine,PencilHolder\WObj:=PAPER;
WaitRob \InPos;
SetDO Do_Kreslit_ON, 0;
SetDO Do_Kreslit_OFF, 1;
MoveL Offs(Target_drawing_origin,-150,50,-5),v100,fine,PencilHolder\WObj:=PAPER;
WaitRob \InPos;
MoveL Offs(Target_drawing_origin,-150,120,-5),v100,fine,PencilHolder\WObj:=PAPER;
WaitRob \InPos;
MoveL Offs(Target_drawing_origin,-150,120,0),v100,fine,PencilHolder\WObj:=PAPER;
WaitRob \InPos;
SetDO Do_Kreslit_ON, 1;
SetDO Do_Kreslit_OFF, 0;
MoveL Offs(Target_drawing_origin,-155,95,0),v100,fine,PencilHolder\WObj:=PAPER;
WaitRob \InPos;
SetDO Do_Kreslit_ON, 0;
SetDO Do_Kreslit_OFF, 1;
MoveL Offs(Target_drawing_origin,-155,95,-5),v100,fine,PencilHolder\WObj:=PAPER;
WaitRob \InPos;
MoveL Offs(Target_drawing_origin,-155,105,-5),v100,fine,PencilHolder\WObj:=PAPER;
WaitRob \InPos;
MoveL Offs(Target_drawing_origin,-155,105,0),v100,fine,PencilHolder\WObj:=PAPER;
WaitRob \InPos;
SetDO Do_Kreslit_ON, 1;
SetDO Do_Kreslit_OFF, 0;
SetDO Do_Kreslit_OFF, 1;


! Draw black
MoveJ Offs(Target_drawing_origin,0,0,-5),v100,fine,PencilHolder\WObj:=PAPER;
MoveL Offs(Target_drawing_origin,-75,15,-5),v100,fine,PencilHolder\WObj:=PAPER;
WaitRob \InPos;
MoveL Offs(Target_drawing_origin,-75,15,0),v100,fine,PencilHolder\WObj:=PAPER;
WaitRob \InPos;
SetDO Do_Kreslit_ON, 1;
SetDO Do_Kreslit_OFF, 0;
MoveL Offs(Target_drawing_origin,-110,15,0),v100,fine,PencilHolder\WObj:=PAPER;
WaitRob \InPos;
SetDO Do_Kreslit_ON, 0;
SetDO Do_Kreslit_OFF, 1;
MoveL Offs(Target_drawing_origin,-110,15,-5),v100,fine,PencilHolder\WObj:=PAPER;
WaitRob \InPos;
MoveL Offs(Target_drawing_origin,-65,20,-5),v100,fine,PencilHolder\WObj:=PAPER;
WaitRob \InPos;
MoveL Offs(Target_drawing_origin,-65,20,0),v100,fine,PencilHolder\WObj:=PAPER;
WaitRob \InPos;
SetDO Do_Kreslit_ON, 1;
SetDO Do_Kreslit_OFF, 0;
MoveL Offs(Target_drawing_origin,-75,20,0),v100,fine,PencilHolder\WObj:=PAPER;
WaitRob \InPos;
SetDO Do_Kreslit_ON, 0;
SetDO Do_Kreslit_OFF, 1;
MoveL Offs(Target_drawing_origin,-75,20,-5),v100,fine,PencilHolder\WObj:=PAPER;
WaitRob \InPos;
MoveL Offs(Target_drawing_origin,-110,20,-5),v100,fine,PencilHolder\WObj:=PAPER;
WaitRob \InPos;
MoveL Offs(Target_drawing_origin,-110,20,0),v100,fine,PencilHolder\WObj:=PAPER;
WaitRob \InPos;
SetDO Do_Kreslit_ON, 1;
SetDO Do_Kreslit_OFF, 0;
MoveL Offs(Target_drawing_origin,-120,20,0),v100,fine,PencilHolder\WObj:=PAPER;
WaitRob \InPos;
SetDO Do_Kreslit_ON, 0;
SetDO Do_Kreslit_OFF, 1;
MoveL Offs(Target_drawing_origin,-120,20,-5),v100,fine,PencilHolder\WObj:=PAPER;
WaitRob \InPos;
MoveL Offs(Target_drawing_origin,-60,25,-5),v100,fine,PencilHolder\WObj:=PAPER;
WaitRob \InPos;
MoveL Offs(Target_drawing_origin,-60,25,0),v100,fine,PencilHolder\WObj:=PAPER;
WaitRob \InPos;
SetDO Do_Kreslit_ON, 1;
SetDO Do_Kreslit_OFF, 0;
MoveL Offs(Target_drawing_origin,-65,25,0),v100,fine,PencilHolder\WObj:=PAPER;
WaitRob \InPos;
SetDO Do_Kreslit_ON, 0;
SetDO Do_Kreslit_OFF, 1;
MoveL Offs(Target_drawing_origin,-65,25,-5),v100,fine,PencilHolder\WObj:=PAPER;
WaitRob \InPos;
MoveL Offs(Target_drawing_origin,-120,25,-5),v100,fine,PencilHolder\WObj:=PAPER;
WaitRob \InPos;
MoveL Offs(Target_drawing_origin,-120,25,0),v100,fine,PencilHolder\WObj:=PAPER;
WaitRob \InPos;
SetDO Do_Kreslit_ON, 1;
SetDO Do_Kreslit_OFF, 0;
MoveL Offs(Target_drawing_origin,-125,25,0),v100,fine,PencilHolder\WObj:=PAPER;
WaitRob \InPos;
SetDO Do_Kreslit_ON, 0;
SetDO Do_Kreslit_OFF, 1;
MoveL Offs(Target_drawing_origin,-125,25,-5),v100,fine,PencilHolder\WObj:=PAPER;
WaitRob \InPos;
MoveL Offs(Target_drawing_origin,-55,30,-5),v100,fine,PencilHolder\WObj:=PAPER;
WaitRob \InPos;
MoveL Offs(Target_drawing_origin,-55,30,0),v100,fine,PencilHolder\WObj:=PAPER;
WaitRob \InPos;
SetDO Do_Kreslit_ON, 1;
SetDO Do_Kreslit_OFF, 0;
MoveL Offs(Target_drawing_origin,-130,30,0),v100,fine,PencilHolder\WObj:=PAPER;
WaitRob \InPos;
SetDO Do_Kreslit_ON, 0;
SetDO Do_Kreslit_OFF, 1;
MoveL Offs(Target_drawing_origin,-130,30,-5),v100,fine,PencilHolder\WObj:=PAPER;
WaitRob \InPos;
MoveL Offs(Target_drawing_origin,-135,30,-5),v100,fine,PencilHolder\WObj:=PAPER;
WaitRob \InPos;
MoveL Offs(Target_drawing_origin,-135,30,0),v100,fine,PencilHolder\WObj:=PAPER;
WaitRob \InPos;
SetDO Do_Kreslit_ON, 1;
SetDO Do_Kreslit_OFF, 0;
MoveL Offs(Target_drawing_origin,-50,35,0),v100,fine,PencilHolder\WObj:=PAPER;
WaitRob \InPos;
SetDO Do_Kreslit_ON, 0;
SetDO Do_Kreslit_OFF, 1;
MoveL Offs(Target_drawing_origin,-50,35,-5),v100,fine,PencilHolder\WObj:=PAPER;
WaitRob \InPos;
MoveL Offs(Target_drawing_origin,-135,35,-5),v100,fine,PencilHolder\WObj:=PAPER;
WaitRob \InPos;
MoveL Offs(Target_drawing_origin,-135,35,0),v100,fine,PencilHolder\WObj:=PAPER;
WaitRob \InPos;
SetDO Do_Kreslit_ON, 1;
SetDO Do_Kreslit_OFF, 0;
MoveL Offs(Target_drawing_origin,-140,35,0),v100,fine,PencilHolder\WObj:=PAPER;
WaitRob \InPos;
SetDO Do_Kreslit_ON, 0;
SetDO Do_Kreslit_OFF, 1;
MoveL Offs(Target_drawing_origin,-140,35,-5),v100,fine,PencilHolder\WObj:=PAPER;
WaitRob \InPos;
MoveL Offs(Target_drawing_origin,-140,40,-5),v100,fine,PencilHolder\WObj:=PAPER;
WaitRob \InPos;
MoveL Offs(Target_drawing_origin,-140,40,0),v100,fine,PencilHolder\WObj:=PAPER;
WaitRob \InPos;
SetDO Do_Kreslit_ON, 1;
SetDO Do_Kreslit_OFF, 0;
MoveL Offs(Target_drawing_origin,-145,45,0),v100,fine,PencilHolder\WObj:=PAPER;
WaitRob \InPos;
SetDO Do_Kreslit_ON, 0;
SetDO Do_Kreslit_OFF, 1;
MoveL Offs(Target_drawing_origin,-145,45,-5),v100,fine,PencilHolder\WObj:=PAPER;
WaitRob \InPos;
MoveL Offs(Target_drawing_origin,-145,50,-5),v100,fine,PencilHolder\WObj:=PAPER;
WaitRob \InPos;
MoveL Offs(Target_drawing_origin,-145,50,0),v100,fine,PencilHolder\WObj:=PAPER;
WaitRob \InPos;
SetDO Do_Kreslit_ON, 1;
SetDO Do_Kreslit_OFF, 0;
MoveL Offs(Target_drawing_origin,-150,60,0),v100,fine,PencilHolder\WObj:=PAPER;
WaitRob \InPos;
SetDO Do_Kreslit_ON, 0;
SetDO Do_Kreslit_OFF, 1;
MoveL Offs(Target_drawing_origin,-150,60,-5),v100,fine,PencilHolder\WObj:=PAPER;
WaitRob \InPos;
MoveL Offs(Target_drawing_origin,-150,65,-5),v100,fine,PencilHolder\WObj:=PAPER;
WaitRob \InPos;
MoveL Offs(Target_drawing_origin,-150,65,0),v100,fine,PencilHolder\WObj:=PAPER;
WaitRob \InPos;
SetDO Do_Kreslit_ON, 1;
SetDO Do_Kreslit_OFF, 0;
MoveL Offs(Target_drawing_origin,-150,70,0),v100,fine,PencilHolder\WObj:=PAPER;
WaitRob \InPos;
SetDO Do_Kreslit_ON, 0;
SetDO Do_Kreslit_OFF, 1;
MoveL Offs(Target_drawing_origin,-150,70,-5),v100,fine,PencilHolder\WObj:=PAPER;
WaitRob \InPos;
MoveL Offs(Target_drawing_origin,-150,75,-5),v100,fine,PencilHolder\WObj:=PAPER;
WaitRob \InPos;
MoveL Offs(Target_drawing_origin,-150,75,0),v100,fine,PencilHolder\WObj:=PAPER;
WaitRob \InPos;
SetDO Do_Kreslit_ON, 1;
SetDO Do_Kreslit_OFF, 0;
MoveL Offs(Target_drawing_origin,-150,80,0),v100,fine,PencilHolder\WObj:=PAPER;
WaitRob \InPos;
SetDO Do_Kreslit_ON, 0;
SetDO Do_Kreslit_OFF, 1;
MoveL Offs(Target_drawing_origin,-150,80,-5),v100,fine,PencilHolder\WObj:=PAPER;
WaitRob \InPos;
MoveL Offs(Target_drawing_origin,-150,85,-5),v100,fine,PencilHolder\WObj:=PAPER;
WaitRob \InPos;
MoveL Offs(Target_drawing_origin,-150,85,0),v100,fine,PencilHolder\WObj:=PAPER;
WaitRob \InPos;
SetDO Do_Kreslit_ON, 1;
SetDO Do_Kreslit_OFF, 0;
MoveL Offs(Target_drawing_origin,-150,90,0),v100,fine,PencilHolder\WObj:=PAPER;
WaitRob \InPos;
SetDO Do_Kreslit_ON, 0;
SetDO Do_Kreslit_OFF, 1;
MoveL Offs(Target_drawing_origin,-150,90,-5),v100,fine,PencilHolder\WObj:=PAPER;
WaitRob \InPos;
MoveL Offs(Target_drawing_origin,-50,170,-5),v100,fine,PencilHolder\WObj:=PAPER;
WaitRob \InPos;
MoveL Offs(Target_drawing_origin,-50,170,0),v100,fine,PencilHolder\WObj:=PAPER;
WaitRob \InPos;
SetDO Do_Kreslit_ON, 1;
SetDO Do_Kreslit_OFF, 0;
MoveL Offs(Target_drawing_origin,-50,175,0),v100,fine,PencilHolder\WObj:=PAPER;
WaitRob \InPos;
SetDO Do_Kreslit_ON, 0;
SetDO Do_Kreslit_OFF, 1;
MoveL Offs(Target_drawing_origin,-50,175,-5),v100,fine,PencilHolder\WObj:=PAPER;
WaitRob \InPos;
MoveL Offs(Target_drawing_origin,-140,175,-5),v100,fine,PencilHolder\WObj:=PAPER;
WaitRob \InPos;
MoveL Offs(Target_drawing_origin,-140,175,0),v100,fine,PencilHolder\WObj:=PAPER;
WaitRob \InPos;
SetDO Do_Kreslit_ON, 1;
SetDO Do_Kreslit_OFF, 0;
SetDO Do_Kreslit_OFF, 1;


ENDPROC


ENDMODULE
